// TIA Portal V17 export
// export: Created 2023-12-22T15:28:32.1014442Z, ExportSetting WithDefaults, DisplayName Totally Integrated Automation Portal, DisplayVersion V17, DisplayName TIA Portal Openness, DisplayVersion V17, DisplayName TIA Portal Version Control Interface, DisplayVersion V17, DisplayName STEP 7 Professional, DisplayVersion V17, DisplayName STEP 7 Safety, DisplayVersion V17, DisplayName WinCC Advanced, DisplayVersion V17
FUNCTION_BLOCK "PLF"   // FB96, LAD
{ S7_Optimized_Access := 'FALSE' }
VERSION : 0.1
// stored: AutoNumber false, IsIECCheckEnabled false, SetENOAutomatically false, UDAEnableTagReadback false
   VAR_INPUT
      Value : Real;   // Показания датчика
   END_VAR
   VAR_IN_OUT
      SP : Real;   // Управляющий сигнал
   END_VAR
   VAR DB_SPECIFIC
      Now : Array[0..10] of Bool;   // Индикатор активного участка
      PLF : Array[0..10] of Struct   // Кусочно-линейная функция
         Use { S7_SetPoint := 'True'} : Bool;   // Использовать участок
         Low : Real;   // Датчик - начальное значение (ось Х)
         High { S7_SetPoint := 'True'} : Real;   // Датчик - конечное значение (ось Х)
         Point_A : Real;   // Управляющий сигнал - минимальное значение (ось Y)
         Point_B { S7_SetPoint := 'True'} : Real;   // Управляющий сигнал - максимальное значение (ось Y)
         res { ExternalAccessible := 'False'; ExternalVisible := 'False'; ExternalWritable := 'False'} : Word;   // резерв
      END_STRUCT;
   END_VAR
   VAR_TEMP   // added for the SCL form of the ladder/FBD networks
      _w1 : Bool;
      _w2 : Bool;
      _w3 : Bool;
      _w4 : Bool;
   END_VAR
BEGIN

REGION Network 1
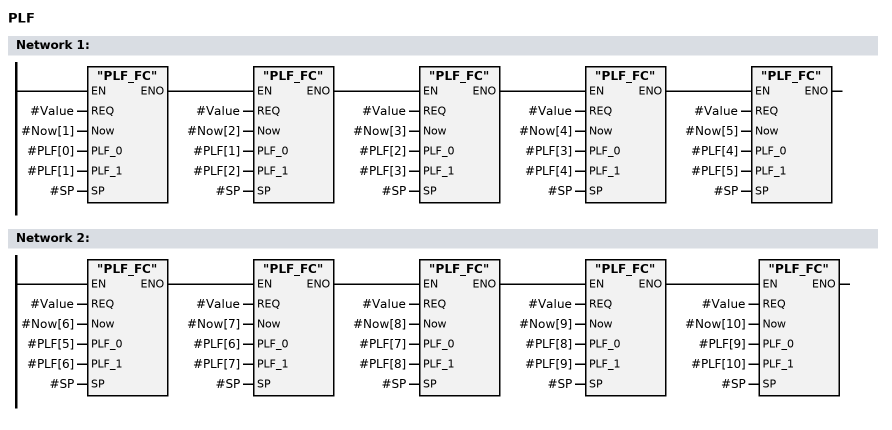
   RUNG wire#powerrail
      "PLF_FC"(REQ := #Value, Now := #Now[1], PLF_0 := #PLF[0], PLF_1 := #PLF[1], SP := #SP)
      "PLF_FC"(REQ := #Value, Now := #Now[2], PLF_0 := #PLF[1], PLF_1 := #PLF[2], SP := #SP)
      "PLF_FC"(REQ := #Value, Now := #Now[3], PLF_0 := #PLF[2], PLF_1 := #PLF[3], SP := #SP)
      "PLF_FC"(REQ := #Value, Now := #Now[4], PLF_0 := #PLF[3], PLF_1 := #PLF[4], SP := #SP)
      "PLF_FC"(REQ := #Value, Now := #Now[5], PLF_0 := #PLF[4], PLF_1 := #PLF[5], SP := #SP)
   END_RUNG
   // the same network as SCL:
   "PLF_FC"(REQ := #Value, Now := #Now[1], PLF_0 := #PLF[0], PLF_1 := #PLF[1], SP := #SP, ENO => #_w1);
   "PLF_FC"(EN := #_w1,
            REQ := #Value,
            Now := #Now[2],
            PLF_0 := #PLF[1],
            PLF_1 := #PLF[2],
            SP := #SP,
            ENO => #_w2);
   "PLF_FC"(EN := #_w2,
            REQ := #Value,
            Now := #Now[3],
            PLF_0 := #PLF[2],
            PLF_1 := #PLF[3],
            SP := #SP,
            ENO => #_w3);
   "PLF_FC"(EN := #_w3,
            REQ := #Value,
            Now := #Now[4],
            PLF_0 := #PLF[3],
            PLF_1 := #PLF[4],
            SP := #SP,
            ENO => #_w4);
   IF #_w4 THEN
       "PLF_FC"(REQ := #Value, Now := #Now[5], PLF_0 := #PLF[4], PLF_1 := #PLF[5], SP := #SP);
   END_IF;
END_REGION

REGION Network 2
   RUNG wire#powerrail
      "PLF_FC"(REQ := #Value, Now := #Now[6], PLF_0 := #PLF[5], PLF_1 := #PLF[6], SP := #SP)
      "PLF_FC"(REQ := #Value, Now := #Now[7], PLF_0 := #PLF[6], PLF_1 := #PLF[7], SP := #SP)
      "PLF_FC"(REQ := #Value, Now := #Now[8], PLF_0 := #PLF[7], PLF_1 := #PLF[8], SP := #SP)
      "PLF_FC"(REQ := #Value, Now := #Now[9], PLF_0 := #PLF[8], PLF_1 := #PLF[9], SP := #SP)
      "PLF_FC"(REQ := #Value, Now := #Now[10], PLF_0 := #PLF[9], PLF_1 := #PLF[10], SP := #SP)
   END_RUNG
   // the same network as SCL:
   "PLF_FC"(REQ := #Value, Now := #Now[6], PLF_0 := #PLF[5], PLF_1 := #PLF[6], SP := #SP, ENO => #_w1);
   "PLF_FC"(EN := #_w1,
            REQ := #Value,
            Now := #Now[7],
            PLF_0 := #PLF[6],
            PLF_1 := #PLF[7],
            SP := #SP,
            ENO => #_w2);
   "PLF_FC"(EN := #_w2,
            REQ := #Value,
            Now := #Now[8],
            PLF_0 := #PLF[7],
            PLF_1 := #PLF[8],
            SP := #SP,
            ENO => #_w3);
   "PLF_FC"(EN := #_w3,
            REQ := #Value,
            Now := #Now[9],
            PLF_0 := #PLF[8],
            PLF_1 := #PLF[9],
            SP := #SP,
            ENO => #_w4);
   IF #_w4 THEN
       "PLF_FC"(REQ := #Value, Now := #Now[10], PLF_0 := #PLF[9], PLF_1 := #PLF[10], SP := #SP);
   END_IF;
END_REGION
END_FUNCTION_BLOCK
